FUNCTION FC_ModeStateToColour : DWORD
VAR_INPUT
	iModeState:INT;
END_VAR
VAR
END_VAR

//converts mode state as integer to colour as DWORD
CASE iModeState OF

//0 = No State
0:
FC_ModeStateToColour := HMIColour.colourWhite;

//1 = Power OFF	
1:
FC_ModeStateToColour := HMIColour.colourWhite;

//2 = Power ON
2:
FC_ModeStateToColour := HMIColour.colourWhite;

//3 = ManualMode
3:
FC_ModeStateToColour := HMIColour.colourWhite;

//4 = AutoMode
4:
FC_ModeStateToColour := HMIColour.colourWhite;

//5 = AutoCycling
5:
FC_ModeStateToColour := HMIColour.colourGreen;

//6 = SemiAuto
6:
FC_ModeStateToColour := HMIColour.colourWhite;

//7 = Fault
7:
FC_ModeStateToColour := HMIColour.colourRed;

//8 = Bypass
8:
FC_ModeStateToColour := HMIColour.colourWhite;

//9 = AutoCycleStopping
9:
FC_ModeStateToColour := HMIColour.colourWhite;

//10 = Dry Cycle
10:
FC_ModeStateToColour := HMIColour.colourWhite;

//11> = spare
11..32767:
FC_ModeStateToColour := HMIColour.colourWhite;




END_CASE

END_FUNCTION

(* stored: Version 1.1.0.1, ProductVersion 3.1.4024.12
   POU FC_ModeStateToColour: Id {7bb523b7-3f37-40a3-a2e4-99638f172644}, SpecialFunc None *)
